// TIA Portal V17 export
// export: Created 2024-09-02T12:50:25.0859079Z, ExportSetting WithDefaults, DisplayName Totally Integrated Automation Portal, DisplayVersion V17, DisplayName TIA Portal Openness, DisplayVersion V17, DisplayName TIA Portal Version Control Interface, DisplayVersion V17, DisplayName STEP 7 Professional, DisplayVersion V17, DisplayName STEP 7 Safety, DisplayVersion V17, DisplayName WinCC Professional, DisplayVersion V17
DATA_BLOCK "Default_SupervisionDB"   // DB8
{ DB_Accessible_From_OPC_UA := 'FALSE' }
VERSION : 0.1
// stored: AutoNumber true, DBAccessibleFromOPCUA false, InstanceOfName Default_SupervisionFB, InstanceOfType FB
"Default_SupervisionFB"
   // VAR
   //    PC_Flags { ExternalWritable := 'False'; S7_SetPoint := 'True'} : PC_Flags_V2;
   //    State { ExternalWritable := 'False'; S7_SetPoint := 'True'} : SV_FB_State_V2;
   //    "AnwDB_ZP_Alarm_OP70.FAULT[1]_I_1" { ExternalWritable := 'False'; S7_SetPoint := 'True'} : SV_State_V2;
   //    "AnwDB_ZP_Alarm_OP70.FAULT[3]_I_1" { ExternalWritable := 'False'; S7_SetPoint := 'True'} : SV_State_V2;
   //    "AnwDB_ZP_Alarm_OP70.FAULT[4]_I_1" { ExternalWritable := 'False'; S7_SetPoint := 'True'} : SV_State_V2;
   //    "AnwDB_ZP_Alarm_OP70.FAULT[5]_I_1" { ExternalWritable := 'False'; S7_SetPoint := 'True'} : SV_State_V2;
   //    "AnwDB_ZP_Alarm_OP70.FAULT[6]_I_1" { ExternalWritable := 'False'; S7_SetPoint := 'True'} : SV_State_V2;
   //    "AnwDB_ZP_Alarm_OP70.FAULT[7]_I_1" { ExternalWritable := 'False'; S7_SetPoint := 'True'} : SV_State_V2;
   //    "AnwDB_ZP_Alarm_OP70.FAULT[8]_I_1" { ExternalWritable := 'False'; S7_SetPoint := 'True'} : SV_State_V2;
   //    "AnwDB_ZP_Alarm_OP70.FAULT[25]_I_1" { ExternalWritable := 'False'; S7_SetPoint := 'True'} : SV_State_V2;
   //    "AnwDB_ZP_Alarm_OP70.FAULT[26]_I_1" { ExternalWritable := 'False'; S7_SetPoint := 'True'} : SV_State_V2;
   //    "AnwDB_ZP_Alarm_OP70.FAULT[27]_I_1" { ExternalWritable := 'False'; S7_SetPoint := 'True'} : SV_State_V2;
   //    "AnwDB_ZP_Alarm_OP70.FAULT[33]_I_1" { ExternalWritable := 'False'; S7_SetPoint := 'True'} : SV_State_V2;
   //    "AnwDB_ZP_Alarm_OP70.FAULT[42]_I_1" { ExternalWritable := 'False'; S7_SetPoint := 'True'} : SV_State_V2;
   //    "AnwDB_ZP_Alarm_OP70.FAULT[45]_I_1" { ExternalWritable := 'False'; S7_SetPoint := 'True'} : SV_State_V2;
   //    "AnwDB_ZP_Alarm_OP70.FAULT[46]_I_1" { ExternalWritable := 'False'; S7_SetPoint := 'True'} : SV_State_V2;
   //    "AnwDB_ZP_Alarm_OP70.FAULT[48]_I_1" { ExternalWritable := 'False'; S7_SetPoint := 'True'} : SV_State_V2;
   //    "AnwDB_ZP_Alarm_OP70.FAULT[49]_I_1" { ExternalWritable := 'False'; S7_SetPoint := 'True'} : SV_State_V2;
   //    "AnwDB_ZP_Alarm_OP70.FAULT[50]_I_1" { ExternalWritable := 'False'; S7_SetPoint := 'True'} : SV_State_V2;
   //    "AnwDB_ZP_Alarm_OP70.FAULT[65]_I_1" { ExternalWritable := 'False'; S7_SetPoint := 'True'} : SV_State_V2;
   //    "AnwDB_ZP_Alarm_OP70.FAULT[66]_I_1" { ExternalWritable := 'False'; S7_SetPoint := 'True'} : SV_State_V2;
   //    "AnwDB_ZP_Alarm_OP70.FAULT[83]_I_1" { ExternalWritable := 'False'; S7_SetPoint := 'True'} : SV_State_V2;
   //    "AnwDB_ZP_Alarm_OP70.FAULT[101]_I_1" { ExternalWritable := 'False'; S7_SetPoint := 'True'} : SV_State_V2;
   //    "AnwDB_ZP_Alarm_OP70.FAULT[102]_I_1" { ExternalWritable := 'False'; S7_SetPoint := 'True'} : SV_State_V2;
   //    "AnwDB_ZP_Alarm_OP70.FAULT[116]_I_1" { ExternalWritable := 'False'; S7_SetPoint := 'True'} : SV_State_V2;
   //    "AnwDB_ZP_Alarm_OP70.FAULT[177]_I_1" { ExternalWritable := 'False'; S7_SetPoint := 'True'} : SV_State_V2;
   //    "AnwDB_ZP_Alarm_OP70.FAULT[178]_I_1" { ExternalWritable := 'False'; S7_SetPoint := 'True'} : SV_State_V2;
   //    "AnwDB_ZP_Alarm_OP70.FAULT[297]_I_1" { ExternalWritable := 'False'; S7_SetPoint := 'True'} : SV_State_V2;
   //    "AnwDB_ZP_Alarm_OP70.FAULT[298]_I_1" { ExternalWritable := 'False'; S7_SetPoint := 'True'} : SV_State_V2;
   //    "AnwDB_ZP_Alarm_OP70.FAULT[299]_I_1" { ExternalWritable := 'False'; S7_SetPoint := 'True'} : SV_State_V2;
   //    "AnwDB_ZP_Alarm_OP70.FAULT[300]_I_1" { ExternalWritable := 'False'; S7_SetPoint := 'True'} : SV_State_V2;
   //    "AnwDB_ZP_Alarm_OP70.FAULT[301]_I_1" { ExternalWritable := 'False'; S7_SetPoint := 'True'} : SV_State_V2;
   //    "AnwDB_ZP_Alarm_OP70.FAULT[302]_I_1" { ExternalWritable := 'False'; S7_SetPoint := 'True'} : SV_State_V2;
   //    "AnwDB_ZP_Alarm_OP70.FAULT[303]_I_1" { ExternalWritable := 'False'; S7_SetPoint := 'True'} : SV_State_V2;
   //    "AnwDB_ZP_Alarm_OP70.FAULT[304]_I_1" { ExternalWritable := 'False'; S7_SetPoint := 'True'} : SV_State_V2;
   //    "AnwDB_ZP_Alarm_OP70.FAULT[305]_I_1" { ExternalWritable := 'False'; S7_SetPoint := 'True'} : SV_State_V2;
   //    "AnwDB_ZP_Alarm_OP70.FAULT[306]_I_1" { ExternalWritable := 'False'; S7_SetPoint := 'True'} : SV_State_V2;
   //    "AnwDB_ZP_Alarm_OP70.FAULT[307]_I_1" { ExternalWritable := 'False'; S7_SetPoint := 'True'} : SV_State_V2;
   //    "AnwDB_ZP_Alarm_OP70.FAULT[308]_I_1" { ExternalWritable := 'False'; S7_SetPoint := 'True'} : SV_State_V2;
   //    "AnwDB_ZP_Alarm_OP70.WARNING[3]_O_1" { ExternalWritable := 'False'; S7_SetPoint := 'True'} : SV_State_V2;
   //    "AnwDB_ZP_Alarm_OP70.WARNING[4]_O_1" { ExternalWritable := 'False'; S7_SetPoint := 'True'} : SV_State_V2;
   //    "AnwDB_ZP_Alarm_OP70.WARNING[5]_O_1" { ExternalWritable := 'False'; S7_SetPoint := 'True'} : SV_State_V2;
   //    "AnwDB_ZP_Alarm_OP70.WARNING[6]_O_1" { ExternalWritable := 'False'; S7_SetPoint := 'True'} : SV_State_V2;
   //    "AnwDB_ZP_Alarm_OP70.WARNING[9]_O_1" { ExternalWritable := 'False'; S7_SetPoint := 'True'} : SV_State_V2;
   //    "AnwDB_ZP_Alarm_OP70.WARNING[20]_O_1" { ExternalWritable := 'False'; S7_SetPoint := 'True'} : SV_State_V2;
   //    "AnwDB_ZP_Alarm_OP70.WARNING[21]_O_1" { ExternalWritable := 'False'; S7_SetPoint := 'True'} : SV_State_V2;
   //    "AnwDB_ZP_Alarm_OP70.WARNING[22]_O_1" { ExternalWritable := 'False'; S7_SetPoint := 'True'} : SV_State_V2;
   //    "AnwDB_ZP_Alarm_OP70.WARNING[23]_O_1" { ExternalWritable := 'False'; S7_SetPoint := 'True'} : SV_State_V2;
   //    "AnwDB_ZP_Alarm_OP70.WARNING[24]_O_1" { ExternalWritable := 'False'; S7_SetPoint := 'True'} : SV_State_V2;
   //    "AnwDB_ZP_Alarm_OP70.WARNING[33]_O_1" { ExternalWritable := 'False'; S7_SetPoint := 'True'} : SV_State_V2;
   //    "AnwDB_ZP_Alarm_OP70.WARNING[34]_O_1" { ExternalWritable := 'False'; S7_SetPoint := 'True'} : SV_State_V2;
   //    "AnwDB_ZP_Alarm_OP70.WARNING[50]_O_1" { ExternalWritable := 'False'; S7_SetPoint := 'True'} : SV_State_V2;
   //    "AnwDB_ZP_Alarm_OP70.WARNING[51]_O_1" { ExternalWritable := 'False'; S7_SetPoint := 'True'} : SV_State_V2;
   //    "AnwDB_ZP_Alarm_OP70.WARNING[110]_O_1" { ExternalWritable := 'False'; S7_SetPoint := 'True'} : SV_State_V2;
   //    "AnwDB_ZP_Alarm_OP70.FAULT[341]_I_1" { ExternalWritable := 'False'; S7_SetPoint := 'True'} : SV_State_V2;
   //    "AnwDB_ZP_Alarm_OP70.FAULT[342]_I_1" { ExternalWritable := 'False'; S7_SetPoint := 'True'} : SV_State_V2;
   //    "AnwDB_ZP_Alarm_OP70.FAULT[343]_I_1" { ExternalWritable := 'False'; S7_SetPoint := 'True'} : SV_State_V2;
   //    "AnwDB_ZP_Alarm_OP70.FAULT[64]_I_1" { ExternalWritable := 'False'; S7_SetPoint := 'True'} : SV_State_V2;
   //    "AnwDB_ZP_Alarm_OP70.FAULT[115]_I_1" { ExternalWritable := 'False'; S7_SetPoint := 'True'} : SV_State_V2;
   //    "AnwDB_ZP_Alarm_OP70.FAULT[344]_I_1" { ExternalWritable := 'False'; S7_SetPoint := 'True'} : SV_State_V2;
   //    "AnwDB_ZP_Alarm_OP70.FAULT[345]_I_1" { ExternalWritable := 'False'; S7_SetPoint := 'True'} : SV_State_V2;
   //    "AnwDB_ZP_Alarm_OP70.FAULT[346]_I_1" { ExternalWritable := 'False'; S7_SetPoint := 'True'} : SV_State_V2;
   //    "AnwDB_ZP_Alarm_OP70.FAULT[347]_I_1" { ExternalWritable := 'False'; S7_SetPoint := 'True'} : SV_State_V2;
   //    "AnwDB_ZP_Alarm_OP70.FAULT[348]_I_1" { ExternalWritable := 'False'; S7_SetPoint := 'True'} : SV_State_V2;
   //    "AnwDB_ZP_Alarm_OP70.FAULT[349]_I_1" { ExternalWritable := 'False'; S7_SetPoint := 'True'} : SV_State_V2;
   //    "AnwDB_ZP_Alarm_OP70.FAULT[350]_I_1" { ExternalWritable := 'False'; S7_SetPoint := 'True'} : SV_State_V2;
   //    "AnwDB_ZP_Alarm_OP70.FAULT[179]_I_1" { ExternalWritable := 'False'; S7_SetPoint := 'True'} : SV_State_V2;
   //    "AnwDB_ZP_Alarm_OP70.FAULT[28]_I_1" { ExternalWritable := 'False'; S7_SetPoint := 'True'} : SV_State_V2;
   //    "AnwDB_ZP_Alarm_OP70.FAULT[180]_I_1" { ExternalWritable := 'False'; S7_SetPoint := 'True'} : SV_State_V2;
   //    "AnwDB_ZP_Alarm_OP70.FAULT[90]_I_1" { ExternalWritable := 'False'; S7_SetPoint := 'True'} : SV_State_V2;
   //    "AnwDB_ZP_Alarm_OP70.FAULT[351]_I_1" { ExternalWritable := 'False'; S7_SetPoint := 'True'} : SV_State_V2;
   //    "AnwDB_ZP_Alarm_OP70.FAULT[352]_I_1" { ExternalWritable := 'False'; S7_SetPoint := 'True'} : SV_State_V2;
   //    "AnwDB_ZP_Alarm_OP70.FAULT[34]_I_1" { ExternalWritable := 'False'; S7_SetPoint := 'True'} : SV_State_V2;
   //    "AnwDB_ZP_Alarm_OP70.WARNING[190]_O_1" { ExternalWritable := 'False'; S7_SetPoint := 'True'} : SV_State_V2;
   //    "AnwDB_ZP_Alarm_OP70.WARNING[191]_O_1" { ExternalWritable := 'False'; S7_SetPoint := 'True'} : SV_State_V2;
   //    "AnwDB_ZP_Alarm_OP70.WARNING[192]_O_1" { ExternalWritable := 'False'; S7_SetPoint := 'True'} : SV_State_V2;
   //    "AnwDB_ZP_Alarm_OP70.FAULT[500]_I_1" { ExternalWritable := 'False'; S7_SetPoint := 'True'} : SV_State_V2;
   //    "AnwDB_ZP_Alarm_OP70.WARNING[300]_O_1" { ExternalWritable := 'False'; S7_SetPoint := 'True'} : SV_State_V2;
   //    "AnwDB_ZP_Alarm_OP70.WARNING[301]_O_1" { ExternalWritable := 'False'; S7_SetPoint := 'True'} : SV_State_V2;
   //    "AnwDB_ZP_Alarm_OP70.FAULT[600]_I_1" { ExternalWritable := 'False'; S7_SetPoint := 'True'} : SV_State_V2;
   //    "AnwDB_ZP_Alarm_OP70.FAULT[601]_I_1" { ExternalWritable := 'False'; S7_SetPoint := 'True'} : SV_State_V2;
   //    "AnwDB_ZP_Alarm_OP70.FAULT[650]_I_1" { ExternalWritable := 'False'; S7_SetPoint := 'True'} : SV_State_V2;
   //    "AnwDB_ZP_Alarm_OP70.FAULT[651]_I_1" { ExternalWritable := 'False'; S7_SetPoint := 'True'} : SV_State_V2;
   //    "AnwDB_ZP_Alarm_OP70.FAULT[700]_I_1" { ExternalWritable := 'False'; S7_SetPoint := 'True'} : SV_State_V2;
   //    "AnwDB_ZP_Alarm_OP70.FAULT[701]_I_1" { ExternalWritable := 'False'; S7_SetPoint := 'True'} : SV_State_V2;
   //    "AnwDB_ZP_Alarm_OP70.FAULT[309]_I_1" { ExternalWritable := 'False'; S7_SetPoint := 'True'} : SV_State_V2;
   //    "AnwDB_ZP_Alarm_OP70.FAULT[310]_I_1" { ExternalWritable := 'False'; S7_SetPoint := 'True'} : SV_State_V2;
   //    "AnwDB_ZP_Alarm_OP70.FAULT[602]_I_1" { ExternalWritable := 'False'; S7_SetPoint := 'True'} : SV_State_V2;
   //    "AnwDB_ZP_Alarm_OP70.FAULT[603]_I_1" { ExternalWritable := 'False'; S7_SetPoint := 'True'} : SV_State_V2;
   //    "AnwDB_ZP_Alarm_OP70.FAULT[604]_I_1" { ExternalWritable := 'False'; S7_SetPoint := 'True'} : SV_State_V2;
   //    "AnwDB_ZP_Alarm_OP70.FAULT[605]_I_1" { ExternalWritable := 'False'; S7_SetPoint := 'True'} : SV_State_V2;
   //    "AnwDB_ZP_Alarm_OP70.FAULT[606]_I_1" { ExternalWritable := 'False'; S7_SetPoint := 'True'} : SV_State_V2;
   //    "AnwDB_ZP_Alarm_OP70.FAULT[607]_I_1" { ExternalWritable := 'False'; S7_SetPoint := 'True'} : SV_State_V2;
   //    "AnwDB_ZP_Alarm_OP70.FAULT[608]_I_1" { ExternalWritable := 'False'; S7_SetPoint := 'True'} : SV_State_V2;
   //    "AnwDB_ZP_Alarm_OP70.FAULT[609]_I_1" { ExternalWritable := 'False'; S7_SetPoint := 'True'} : SV_State_V2;
   //    "AnwDB_ZP_Alarm_OP70.FAULT[610]_I_1" { ExternalWritable := 'False'; S7_SetPoint := 'True'} : SV_State_V2;
   //    "AnwDB_ZP_Alarm_OP70.FAULT[611]_I_1" { ExternalWritable := 'False'; S7_SetPoint := 'True'} : SV_State_V2;
   //    "AnwDB_ZP_Alarm_OP70.FAULT[612]_I_1" { ExternalWritable := 'False'; S7_SetPoint := 'True'} : SV_State_V2;
   //    "AnwDB_ZP_Alarm_OP70.FAULT[613]_I_1" { ExternalWritable := 'False'; S7_SetPoint := 'True'} : SV_State_V2;
   //    "AnwDB_ZP_Alarm_OP70.FAULT[614]_I_1" { ExternalWritable := 'False'; S7_SetPoint := 'True'} : SV_State_V2;
   //    "AnwDB_ZP_Alarm_OP70.FAULT[615]_I_1" { ExternalWritable := 'False'; S7_SetPoint := 'True'} : SV_State_V2;
   //    "AnwDB_ZP_Alarm_OP70.FAULT[616]_I_1" { ExternalWritable := 'False'; S7_SetPoint := 'True'} : SV_State_V2;
   //    "AnwDB_ZP_Alarm_OP70.FAULT[617]_I_1" { ExternalWritable := 'False'; S7_SetPoint := 'True'} : SV_State_V2;
   //    "AnwDB_ZP_Alarm_OP70.FAULT[618]_I_1" { ExternalWritable := 'False'; S7_SetPoint := 'True'} : SV_State_V2;
   //    "AnwDB_ZP_Alarm_OP70.FAULT[800]_I_1" { ExternalWritable := 'False'; S7_SetPoint := 'True'} : SV_State_V2;
   //    "AnwDB_ZP_Alarm_OP70.WARNING[302]_O_1" { ExternalWritable := 'False'; S7_SetPoint := 'True'} : SV_State_V2;
   //    "AnwDB_ZP_Alarm_OP70.WARNING[303]_O_1" { ExternalWritable := 'False'; S7_SetPoint := 'True'} : SV_State_V2;
   //    "AnwDB_ZP_Alarm_OP70.WARNING[304]_O_1" { ExternalWritable := 'False'; S7_SetPoint := 'True'} : SV_State_V2;
   //    "AnwDB_ZP_Alarm_OP70.WARNING[305]_O_1" { ExternalWritable := 'False'; S7_SetPoint := 'True'} : SV_State_V2;
   //    "AnwDB_ZP_Alarm_OP70.WARNING[306]_O_1" { ExternalWritable := 'False'; S7_SetPoint := 'True'} : SV_State_V2;
   //    "AnwDB_ZP_Alarm_OP70.WARNING[307]_O_1" { ExternalWritable := 'False'; S7_SetPoint := 'True'} : SV_State_V2;
   // END_VAR
BEGIN
END_DATA_BLOCK
